FUNCTION_BLOCK DT_TO_DOY_UINT (* Composite Function Block Type *)
  (* Standard: 61499-2 *)
  (* Version 0.0, 2017-06-05, 4DIAC-IDE, 4DIAC-Consortium *)
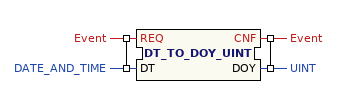
  EVENT_INPUT
    REQ WITH DT; (* Normal Execution Request *)
  END_EVENT
  EVENT_OUTPUT
    CNF WITH DOY; (* Execution Confirmation *)
  END_EVENT
  VAR_INPUT
    DT : DATE_AND_TIME; (* Input date *)
  END_VAR
  VAR_OUTPUT
    DOY : UINT; (* Output event qualifier *)
  END_VAR
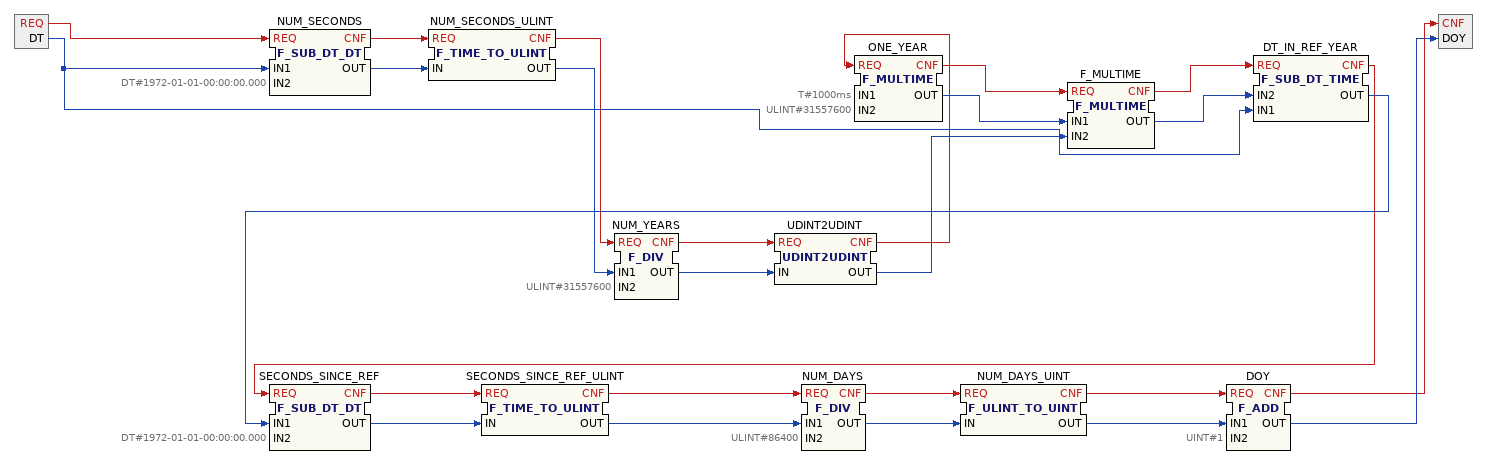
  FBS
    NUM_SECONDS : F_SUB_DT_DT(IN2 := DT#1972-01-01-00:00:00.000);
    NUM_SECONDS_ULINT : F_TIME_TO_ULINT;
    NUM_YEARS : F_DIV(IN2 := ULINT#31557600);
    F_MULTIME : F_MULTIME;
    DT_IN_REF_YEAR : F_SUB_DT_TIME;
    SECONDS_SINCE_REF_ULINT : F_TIME_TO_ULINT;
    SECONDS_SINCE_REF : F_SUB_DT_DT(IN2 := DT#1972-01-01-00:00:00.000);
    ONE_YEAR : F_MULTIME(IN1 := T#1000ms, IN2 := ULINT#31557600);
    NUM_DAYS : F_DIV(IN2 := ULINT#86400);
    NUM_DAYS_UINT : F_ULINT_TO_UINT;
    DOY : F_ADD(IN2 := UINT#1);
    UDINT2UDINT : UDINT2UDINT;
  END_FBS
  EVENT_CONNECTIONS
    NUM_SECONDS.CNF TO NUM_SECONDS_ULINT.REQ;
    REQ TO NUM_SECONDS.REQ;
    NUM_SECONDS_ULINT.CNF TO NUM_YEARS.REQ;
    F_MULTIME.CNF TO DT_IN_REF_YEAR.REQ;
    ONE_YEAR.CNF TO F_MULTIME.REQ;
    SECONDS_SINCE_REF_ULINT.CNF TO NUM_DAYS.REQ;
    NUM_DAYS.CNF TO NUM_DAYS_UINT.REQ;
    NUM_DAYS_UINT.CNF TO DOY.REQ;
    DOY.CNF TO CNF;
    NUM_YEARS.CNF TO UDINT2UDINT.REQ;
    UDINT2UDINT.CNF TO ONE_YEAR.REQ;
    DT_IN_REF_YEAR.CNF TO SECONDS_SINCE_REF.REQ;
    SECONDS_SINCE_REF.CNF TO SECONDS_SINCE_REF_ULINT.REQ;
  END_CONNECTIONS
  DATA_CONNECTIONS
    NUM_SECONDS.OUT TO NUM_SECONDS_ULINT.IN;
    DT TO NUM_SECONDS.IN1;
    NUM_SECONDS_ULINT.OUT TO NUM_YEARS.IN1;
    F_MULTIME.OUT TO DT_IN_REF_YEAR.IN2;
    DT TO DT_IN_REF_YEAR.IN1;
    ONE_YEAR.OUT TO F_MULTIME.IN1;
    SECONDS_SINCE_REF_ULINT.OUT TO NUM_DAYS.IN1;
    NUM_DAYS.OUT TO NUM_DAYS_UINT.IN;
    NUM_DAYS_UINT.OUT TO DOY.IN1;
    DOY.OUT TO DOY;
    NUM_YEARS.OUT TO UDINT2UDINT.IN;
    UDINT2UDINT.OUT TO F_MULTIME.IN2;
    DT_IN_REF_YEAR.OUT TO SECONDS_SINCE_REF.IN1;
    SECONDS_SINCE_REF.OUT TO SECONDS_SINCE_REF_ULINT.IN;
  END_CONNECTIONS
END_FUNCTION_BLOCK
